// TIA Portal V17 export
// export: Created 2023-12-22T15:04:42.4152447Z, ExportSetting WithDefaults, DisplayName Totally Integrated Automation Portal, DisplayVersion V17, DisplayName TIA Portal Openness, DisplayVersion V17, DisplayName TIA Portal Version Control Interface, DisplayVersion V17, DisplayName STEP 7 Professional, DisplayVersion V17, DisplayName STEP 7 Safety, DisplayVersion V17, DisplayName WinCC Advanced, DisplayVersion V17
DATA_BLOCK "PID_Flow_DB"   // DB900
VERSION : 0.1
// stored: AutoNumber false, DBAccessibleFromOPCUA true, InstanceOfName PID_ex, InstanceOfType FB
"PID_ex"
   // VAR_INPUT
   //    Start : Bool;
   //    SP_A : Real;
   //    Value : Real;
   // END_VAR
   // VAR_OUTPUT
   //    PWM : Bool;
   //    Result : Real;
   // END_VAR
   // VAR RETAIN
   //    CMD { S7_SetPoint := 'True'} : "CMD";
   //    SP_M : Real;
   //    SP : Real;
   //    x { S7_SetPoint := 'True'} : Real := 1.0;
   //    SP_x : Real;
   //    Value_x : Real;
   //    Buffer : Real;
   //    PID_Output : Real;
   //    PID_Hand : Real;
   //    Sys : Struct
   //       Err_Ack : Bool;
   //       Alm_SP_H : Bool;
   //       Alm_SP_L : Bool;
   //       Alm_In_H : Bool;
   //       Alm_In_L : Bool;
   //       Activate : Bool;
   //       Error_code : DWord;
   //       Warning_code : DWord;
   //       "Type" : Int;
   //       State : Int;
   //       Mode : Int;
   //    END_STRUCT;
   //    Settings : Struct
   //       SP_P { S7_SetPoint := 'True'} : Real := 1.5;
   //       SP_Ti { S7_SetPoint := 'True'} : Real := 150.0;
   //       SP_Td { S7_SetPoint := 'True'} : Real := 0.0;
   //       SP_Cycle { S7_SetPoint := 'True'} : Real := 0.2;
   //       Max_SP { S7_SetPoint := 'True'} : Real := 500.0;
   //       Min_SP { S7_SetPoint := 'True'} : Real := -500.0;
   //       Max_in { S7_SetPoint := 'True'} : Real := 500.0;
   //       Min_in { S7_SetPoint := 'True'} : Real := -500.0;
   //       Max_out { S7_SetPoint := 'True'} : Real := 100.0;
   //       Min_out { S7_SetPoint := 'True'} : Real := 0.0;
   //       DeadBand { S7_SetPoint := 'True'} : Real := 1.0;
   //       Max : Real;
   //       Min : Real;
   //    END_STRUCT;
   //    PID { S7_SetPoint := 'True'} : PID_Compact;
   //    Converter : "Converter_SCL";
   //    Conveter_Back : "Converter_SCL";
   //    C { S7_SetPoint := 'True'} : "Time_R";
   //    pos : Array[0..15] of Bool;
   // END_VAR
BEGIN
   CMD.Vector := FALSE;
   PID.IntegralResetMode := 4;
   PID.RunModeByStartup := TRUE;
   PID.SetSubstituteOutput := TRUE;
   PID.ActivateRecoverMode := TRUE;
   PID.CancelTuningLevel := 10.0;
   PID.SubstituteOutput := 0.0;
   PID.Config.InputPerOn := FALSE;
   PID.Config.InvertControl := FALSE;
   PID.Config.InputUpperLimit := 500.0;
   PID.Config.InputLowerLimit := -500.0;
   PID.Config.InputUpperWarning := 3.402822E+38;
   PID.Config.InputLowerWarning := -3.402822E+38;
   PID.Config.OutputUpperLimit := 100.0;
   PID.Config.OutputLowerLimit := 0.0;
   PID.Config.SetpointUpperLimit := 500.0;
   PID.Config.SetpointLowerLimit := -500.0;
   PID.Config.MinimumOnTime := 0.0;
   PID.Config.MinimumOffTime := 0.0;
   PID.Config.InputScaling.UpperPointIn := 27648.0;
   PID.Config.InputScaling.LowerPointIn := 0.0;
   PID.Config.InputScaling.UpperPointOut := 100.0;
   PID.Config.InputScaling.LowerPointOut := 0.0;
   PID.CycleTime.EnEstimation := TRUE;
   PID.CycleTime.EnMonitoring := TRUE;
   PID.CycleTime.Value := 0.1;
   PID.CtrlParamsBackUp.Gain := 1.0;
   PID.CtrlParamsBackUp.Ti := 20.0;
   PID.CtrlParamsBackUp.Td := 0.0;
   PID.CtrlParamsBackUp.TdFiltRatio := 0.2;
   PID.CtrlParamsBackUp.PWeighting := 1.0;
   PID.CtrlParamsBackUp.DWeighting := 1.0;
   PID.CtrlParamsBackUp.Cycle := 1.0;
   PID.PIDSelfTune.SUT.TuneRule := 1;
   PID.PIDSelfTune.TIR.TuneRule := 0;
   PID.Retain.CtrlParams.Gain := 1.5;
   PID.Retain.CtrlParams.Ti := 150.0;
   PID.Retain.CtrlParams.Td := 0.0;
   PID.Retain.CtrlParams.TdFiltRatio := 0.2;
   PID.Retain.CtrlParams.PWeighting := 1.0;
   PID.Retain.CtrlParams.DWeighting := 1.0;
   PID.Retain.CtrlParams.Cycle := 1.0;
   C.SP := 0.2;
   C.One := 0.1;
END_DATA_BLOCK
